PROGRAM MachineSimulation
VAR
    fbMachine	:	FB_MachineSimulator; //Simulates attenuator as well
    fbeVSimulator : FB_eVSimulator := (NoiseLevel := 1);
END_VAR

// reV Simulator
fbeVSimulator();

// Machine simulator
fbMachine(
    i_stAssertedParams := PMPS_GVL.stRequestedBeamParameters,
    q_stMachineParams => PMPS_GVL.stCurrentBeamParameters,
    i_xFault	:= NOT GVL.g_FastFaultOutput1.q_xFastFaultOut
    );

PMPS_GVL.stCurrentBeamParameters.neVRange := F_eVRangeCalculator(fbeVSimulator.eV, PMPS_GVL.stCurrentBeamParameters.neVRange);

END_PROGRAM

(* stored: Version 1.1.0.1, ProductVersion 3.1.4022.18
   POU MachineSimulation: Id {215532fb-b2c1-07b9-12dd-bf8b9df2fcb5}, SpecialFunc None *)
